{attribute 'linkalways'} 
{attribute 'no_explicit_call' := 'This FB is a CLASS and must be accessed using methods or properties'}
{attribute 'enable_dynamic_creation'}
FUNCTION_BLOCK _ETcVnColorTrainingMethod EXTENDS EnumDatatypeBase
VAR
	localData : ETcVnColorTrainingMethod;
	activeData : REFERENCE TO ETcVnColorTrainingMethod;
	enumBaseDatatype : _DINT(localData);
END_VAR

METHOD PRIVATE AddLocalEnumeration
VAR_INPUT
	Enumeration : T_MAXSTRING;
	Value : ETcVnColorTrainingMethod;
END_VAR
AddEnumeration(Enumeration, Value);
END_METHOD

PROPERTY PUBLIC Address : PVOID
GET
Address := ADR(activeData);
END_GET
END_PROPERTY

METHOD PUBLIC ClearReference
VAR_INPUT
END_VAR
activeData REF= localData;
SetBaseDatatypeReference();
END_METHOD

METHOD PUBLIC Clone : I_Datatype
VAR
    pClone : POINTER TO _ETcVnColorTrainingMethod;
END_VAR
pClone := __NEW(_ETcVnColorTrainingMethod(InitialValue := Value));
Clone := pClone^;
END_METHOD

METHOD FB_init : BOOL
VAR_INPUT
	bInitRetains : BOOL; // if TRUE, the retain variables are initialized (warm start / cold start)
	bInCopyCode : BOOL;  // if TRUE, the instance afterwards gets moved into the copy code (online change)
	InitialValue : ETcVnColorTrainingMethod;
END_VAR
localData := InitialValue;
AddBaseDatatype(enumBaseDatatype);
ClearReference();

AddLocalEnumeration('TCVN_CTM_LAB', ETcVnColorTrainingMethod.TCVN_CTM_LAB);
AddLocalEnumeration('TCVN_CTM_RGB', ETcVnColorTrainingMethod.TCVN_CTM_RGB);
END_METHOD

PROPERTY PUBLIC Identifier : T_MAXSTRING
GET
Identifier := 'ETcVnColorTrainingMethod';
END_GET
END_PROPERTY

METHOD IsEnumeratorValueEqual : BOOL
VAR_INPUT
	Enumerator : I_KeyValueForwardEnumerator;
END_VAR
VAR
	storedValue : ETcVnColorTrainingMethod;
END_VAR
IF NOT Enumerator.TryGet(storedValue) THEN
	RETURN;
END_IF

IsEnumeratorValueEqual := storedValue = activeData;
END_METHOD

METHOD PUBLIC MakeReferenceTo
VAR_INPUT
	ReferenceTarget : REFERENCE TO ETcVnColorTrainingMethod;
END_VAR
activeData REF= ReferenceTarget;
SetBaseDatatypeReference();
END_METHOD

METHOD PROTECTED SetBaseDatatypeReference
VAR_INPUT
END_VAR
enumBaseDatatype.MakeReferenceTo(activeData);
END_METHOD

PROPERTY PUBLIC Size : UDINT
GET
Size := SIZEOF(activeData);
END_GET
END_PROPERTY

METHOD TryMakeReferenceTo : BOOL
VAR_INPUT
	Target : I_Datatype;
END_VAR
VAR
	targetAsEnum : I_EnumDatatype;
	pTargetData : POINTER TO ETcVnColorTrainingMethod;
END_VAR
IF NOT Target.TryResolveAsEnumDatatype(targetAsEnum) THEN
	RETURN;
END_IF

IF targetAsEnum.Identifier <> Identifier THEN
	RETURN;
END_IF

pTargetData := Target.Address;
activeData REF= pTargetData^;
SetBaseDatatypeReference();
TryMakeReferenceTo := TRUE;
END_METHOD

PROPERTY PUBLIC Value : ETcVnColorTrainingMethod
GET
Value := activeData;
END_GET
SET
activeData := Value;
END_SET
END_PROPERTY

END_FUNCTION_BLOCK

(* stored: Version 1.1.0.1, ProductVersion 3.1.4024.12
   POU _ETcVnColorTrainingMethod: Id {fa23e47b-d9af-44e7-9d2e-de8623e4e651}, SpecialFunc None
   Folder Constructor: Id {81b8b4a0-b91b-462b-8a91-d5290b536aad}
   Folder Private: Id {551abea1-3d79-4338-9904-fe49e9dbff06}
   Folder Protected: Id {6b1c661f-5231-48bc-8be8-48685ff9d476}
   Method AddLocalEnumeration: Id {2de8daa3-8ba1-4fd8-8abe-7d51dfb059ab}
   Property Address: Id {2c8935f7-1e1b-4df6-95b1-f4a50b42725b}
   Get Get: Id {00dc3b87-3814-4ab3-bdb8-2a0dc197fff6}
   Method ClearReference: Id {f984b7dc-5c17-4c9d-bfa3-15fa158f0702}
   Method Clone: Id {18d0541d-a4ea-4acb-a363-9a1fc8fbd563}
   Method FB_init: Id {af8bc4f3-f40e-4190-a808-32f64162b3ae}
   Property Identifier: Id {951faab8-b2de-43ac-a93c-4e299750fba5}
   Get Get: Id {e431cc16-0533-4dc7-899a-4e87c42cf331}
   Method IsEnumeratorValueEqual: Id {c416eacd-1169-44d4-9811-9947461cc77f}
   Method MakeReferenceTo: Id {7664a061-cca4-44e5-8f9d-b6d1b6ea4aea}
   Method SetBaseDatatypeReference: Id {ec6b3adc-25ab-4399-8664-3d5dac3a6336}
   Property Size: Id {087fc1e6-86be-4f44-ac2f-61c93140bc73}
   Get Get: Id {827c92d1-e1a9-45b9-97d1-3923fec6e391}
   Method TryMakeReferenceTo: Id {66a22d50-205b-41e5-b42e-1ae4b449d6d8}
   Property Value: Id {157ebaed-8b82-41b4-a70b-0e92f7d37f36}
   Get Get: Id {cdeaa89a-3276-46a9-9192-eb216237515e}
   Set Set: Id {00633535-d2b3-4bff-ac5a-0c9bb4eef1e2} *)
